# EPICS autosave request: autosave/galil_coordinate_system.req
$(P)$(R)_STOP_CMD
$(P)$(R)_GO_CMD
